{attribute 'GeneratedUsingTerminal: EJ7031-0000-0026'}
{attribute addProperty BoxType "EJ7031-0000-0026"}
{attribute addProperty Id "VelocityAT %Q*INT2"}
{attribute addProperty CRC "2759475009"}
{attribute addProperty Size "2"}
TYPE STM_Velocity_A47A3F41 :
STRUCT
	{attribute addProperty Name "Velocity"}
	Velocity AT %Q* : INT;
END_STRUCT
END_TYPE

(* stored: Version 1.2.0.0, ProductVersion 3.1.4024.9
   DUT STM_Velocity_A47A3F41: Id {49e379d9-0c9b-4b63-8c5f-b5925cb4588d} *)
